FUNCTION_BLOCK SHIFT_ANY (* Abstract superclass for IEC 61131-3 bit shift functions *)
  (* Standard: 61131-3 *)
  (* Version 0.0, 2004-12-15, JHC, Rockwell Automation, Converted from SRC format. *)
  (* Compiler header: package fb.rt.plc.bits; *)
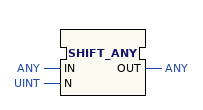
  VAR_INPUT
    IN : ANY; (* ANY_BIT to be shifted *)
    N : UINT; (* Shift count *)
  END_VAR
  VAR_OUTPUT
    OUT : ANY; (* Value of IN shifted N bits *)
  END_VAR
END_FUNCTION_BLOCK
